TYPE ST_Vis_ControlPadControl :
STRUCT
	
	bVisInvisibleButton	: BOOL;	
	bVisInvisible		: BOOL;	
	nFramePositionX		: INT;
	nFramePositionY		: INT;
	nButtonPositionX	: INT;
	nButtonPositionY	: INT;
	
	bButtonState_Abort			: BOOL;
	bButtonState_Reset			: BOOL;
	bButtonState_Prepare		: BOOL;	
	bButtonState_Start			: BOOL;
	
	bStateSignalAbortBlue		: BOOL;
	bStateSignalAbortYellow		: BOOL;
	bStateSignalAbortGreen		: BOOL;
	
	bStateSignalResetYellow		: BOOL;
	bStateSignalResetGreen		: BOOL;

	bStateSignalPrepareYellow	: BOOL;
	bStateSignalPrepareGreen	: BOOL;

	bStateSignalExecuteYellow	: BOOL;
	bStateSignalExecuteGreen	: BOOL;	

	bAbortSequenceStateInvisible	: BOOL;
	bResetSequenceStateInvisible	: BOOL;
	bPrepareSequenceStateInvisible	: BOOL;
	bStartSequenceStateInvisible	: BOOL;
	
	iAbortSequenceState			: INT;
	iResetSequenceState			: INT;
	iPrepareSequenceState		: INT;
	iStartSequenceState			: INT;	
	
	
END_STRUCT
END_TYPE

(* stored: Version 1.1.0.1, ProductVersion 3.1.4024.4
   DUT ST_Vis_ControlPadControl: Id {b518f074-0dbe-4ce1-984a-c052d3942081} *)
